Staubli VAL3: onStart.pgx

program onStart()
  local num i
begin
  // logMsg
  logMsg("[KERNEL] INTERFACE:PAGE Process List")
  // reset the Key pressure
  call use:nullKey(nKey)
  // define the list
  call buildList()
  // build the page
  call refreshStatic()
  //
end
